SUBAPPLICATION Speed_Selection (* Waehlt aus den verfuegbaren Geschwindigkeitssignalen (VDS, WBSD, GBSD, MSS) das vom Bediener ausgewaehlte Signal aus und stellt Geschwindigkeit, Richtung und zurueckgelegte Distanz bereit; die Auswahl wird persistent im NVS gespeichert *)
  (* Standard: 61499-2 *)
  (* Version 1.0, 2025-04-01, Elias *)
  PACKAGE FBs::Baumsetzer::func::Automatik;
  IMPORT NVS_Keys::Key_GBSD_Store;
  IMPORT NVS_Keys::Key_MSS_Store;
  IMPORT NVS_Keys::Key_NMEA_Store;
  IMPORT NVS_Keys::Key_VDS_Store;
  IMPORT NVS_Keys::Key_WBSD_Store;
  IMPORT isobus::UT::Q::const::colours::COLOR_GREEN;
  IMPORT isobus::UT::Q::const::colours::COLOR_RED;
  IMPORT isobus::UT::io::Button::ButtonActivationCode::BT_RELEASED_UNLATCHED;
  IMPORT test::FBs::Baumsetzer::Constants::DefaultPool;
  IMPORT test::FBs::Baumsetzer::Constants::DefaultPool::Button_GBSD;
  IMPORT test::FBs::Baumsetzer::Constants::DefaultPool::Button_MSS;
  IMPORT test::FBs::Baumsetzer::Constants::DefaultPool::Button_NMEA;
  IMPORT test::FBs::Baumsetzer::Constants::DefaultPool::Button_VDS;
  IMPORT test::FBs::Baumsetzer::Constants::DefaultPool::Button_WBSD;
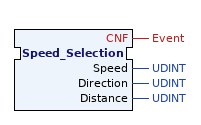
  EVENT_OUTPUT
    CNF; (* Execution Confirmation *)
  END_EVENT
  VAR_OUTPUT
    Speed : UDINT; (* Speed of selected Signal *)
    Direction : UDINT; (* Direction of selected Signal *)
    Distance : UDINT; (* Distance of selected Signal *)
  END_VAR
  FBS
    I_MSS : isobus::tecu::I_MSS(QI := FALSE);
    I_GBSD : isobus::tecu::I_GBSD(QI := FALSE);
    I_WBSD : isobus::tecu::I_WBSD(QI := FALSE);
    I_VDS : isobus::tecu::I_VDS(QI := FALSE);
    Button_VDS : isobus::UT::io::Button::Button_IE(QI := TRUE, u16ObjId := Button_VDS, InputEvent := BT_RELEASED_UNLATCHED);
    Button_WBSD : isobus::UT::io::Button::Button_IE(QI := TRUE, PARAMS := '', u16ObjId := Button_WBSD, InputEvent := BT_RELEASED_UNLATCHED);
    Button_GBSD : isobus::UT::io::Button::Button_IE(QI := TRUE, u16ObjId := Button_GBSD, InputEvent := BT_RELEASED_UNLATCHED);
    Button_MSS : isobus::UT::io::Button::Button_IE(QI := TRUE, u16ObjId := Button_MSS, InputEvent := BT_RELEASED_UNLATCHED);
    F_UINT_TO_REAL : iec61131::conversion::F_UINT_TO_REAL;
    CYCLE_TIME : logiBUS::utils::timing::CYCLE_TIME;
    INTEGRAL : logiBUS::utils::math::INTEGRAL;
    E_T_FF_SR : iec61499::events::E_T_FF_SR;
    E_T_FF_SR_1 : iec61499::events::E_T_FF_SR;
    E_T_FF_SR_2 : iec61499::events::E_T_FF_SR;
    E_T_FF_SR_3 : iec61499::events::E_T_FF_SR;
    F_SEL_E_Distance : eclipse4diac::utils::selection::F_SEL_E_4;
    F_SEL_E_Speed : eclipse4diac::utils::selection::F_SEL_E_4;
    F_SEL_E_Direction : eclipse4diac::utils::selection::F_SEL_E_4;
    COGSOGRapidUpdate : isobus::tecu::I_COGSOGRapidUpdate;
    E_T_FF_SR_4 : iec61499::events::E_T_FF_SR;
    Button_NMEA : isobus::UT::io::Button::Button_IE(QI := TRUE, u16ObjId := Button_NMEA, InputEvent := BT_RELEASED_UNLATCHED);
    INTEGRAL_1 : logiBUS::utils::math::INTEGRAL;
    CYCLE_TIME_1 : logiBUS::utils::timing::CYCLE_TIME;
    F_UINT_TO_REAL_1 : iec61131::conversion::F_UINT_TO_REAL;
    F_SEL_E_Distance_2 : eclipse4diac::utils::selection::F_SEL_E_2;
    F_SEL_E_Speed_2 : eclipse4diac::utils::selection::F_SEL_E_2;
    F_SEL_E_Direction_2 : eclipse4diac::utils::selection::F_SEL_E_2;
    UDINT2UDINT : iec61131::selection::F_MOVE; {SET_ATTRIBUTE(DataType, UDINT)}
    UDINT2UDINT_1 : iec61131::selection::F_MOVE; {SET_ATTRIBUTE(DataType, UDINT)}
    UDINT2UDINT_2 : iec61131::selection::F_MOVE; {SET_ATTRIBUTE(DataType, UDINT)}
    E_PERMIT : iec61499::events::E_PERMIT;
    E_PERMIT_1 : iec61499::events::E_PERMIT;
    E_PERMIT_2 : iec61499::events::E_PERMIT;
    E_PERMIT_4 : iec61499::events::E_PERMIT;
    F_SEL : iec61131::selection::F_SEL(IN0 := COLOR_RED, IN1 := COLOR_GREEN);
    Q_BackgroundColour : isobus::UT::Q::Q_BackgroundColour(u16ObjId := Button_VDS);
    Q_BackgroundColour_1 : isobus::UT::Q::Q_BackgroundColour(u16ObjId := Button_WBSD);
    F_SEL_1 : iec61131::selection::F_SEL(IN0 := COLOR_RED, IN1 := COLOR_GREEN);
    Q_BackgroundColour_2 : isobus::UT::Q::Q_BackgroundColour(u16ObjId := Button_GBSD);
    F_SEL_2 : iec61131::selection::F_SEL(IN0 := COLOR_RED, IN1 := COLOR_GREEN);
    Q_BackgroundColour_3 : isobus::UT::Q::Q_BackgroundColour(u16ObjId := Button_MSS);
    F_SEL_3 : iec61131::selection::F_SEL(IN0 := COLOR_RED, IN1 := COLOR_GREEN);
    Q_BackgroundColour_4 : isobus::UT::Q::Q_BackgroundColour(u16ObjId := Button_NMEA);
    F_SEL_4 : iec61131::selection::F_SEL(IN0 := COLOR_RED, IN1 := COLOR_GREEN);
    Geschwindigkeit : isobus::UT::Q::Q_NumericValue(u16ObjId := DefaultPool::OutputNumber_12000);
    Geschwindigkeit_1 : isobus::UT::Q::Q_NumericValue(u16ObjId := DefaultPool::OutputNumber_12004);
    Geschwindigkeit_2 : isobus::UT::Q::Q_NumericValue(u16ObjId := DefaultPool::OutputNumber_12005);
    Geschwindigkeit_3 : isobus::UT::Q::Q_NumericValue(u16ObjId := DefaultPool::OutputNumber_12006);
    Geschwindigkeit_4 : isobus::UT::Q::Q_NumericValue(u16ObjId := DefaultPool::OutputNumber_12007);
    F_MUL : iec61131::arithmetic::F_MUL(IN2 := uint#10);
    CYCLE_TIME_2 : logiBUS::utils::timing::CYCLE_TIME;
    E_PERMIT_5 : iec61499::events::E_PERMIT;
    INTEGRAL_2 : logiBUS::utils::math::INTEGRAL;
    F_UINT_TO_REAL_2 : iec61131::conversion::F_UINT_TO_REAL;
    F_REAL_TO_UDINT : iec61131::conversion::F_REAL_TO_UDINT;
    F_REAL_TO_UDINT_1 : iec61131::conversion::F_REAL_TO_UDINT;
    F_REAL_TO_UDINT_2 : iec61131::conversion::F_REAL_TO_UDINT;
    UDINT2UDINT_Distance : iec61131::selection::F_MOVE; {SET_ATTRIBUTE(DataType, UDINT)}
    UDINT2UDINT_Speed : iec61131::selection::F_MOVE; {SET_ATTRIBUTE(DataType, UDINT)}
    UDINT2UDINT_Direction : iec61131::selection::F_MOVE; {SET_ATTRIBUTE(DataType, UDINT)}
    VDS_Selected : logiBUS::storage::esp32_nvs::NVS(QI := TRUE, KEY := Key_VDS_Store, DEFAULT_VALUE := bool#FALSE);
    WBSD_Selected : logiBUS::storage::esp32_nvs::NVS(QI := TRUE, KEY := Key_WBSD_Store, DEFAULT_VALUE := bool#TRUE);
    GBSD_Selected : logiBUS::storage::esp32_nvs::NVS(QI := TRUE, KEY := Key_GBSD_Store, DEFAULT_VALUE := bool#FALSE);
    F_MOVE_2 : iec61131::selection::F_MOVE; {SET_ATTRIBUTE(DataType, BOOL)}
    MSS_Selected : logiBUS::storage::esp32_nvs::NVS(QI := TRUE, KEY := Key_MSS_Store, DEFAULT_VALUE := bool#FALSE);
    F_MOVE_3 : iec61131::selection::F_MOVE; {SET_ATTRIBUTE(DataType, BOOL)}
    NMEA_Selected : logiBUS::storage::esp32_nvs::NVS(QI := TRUE, KEY := Key_NMEA_Store, DEFAULT_VALUE := bool#FALSE);
    F_MOVE_4 : iec61131::selection::F_MOVE; {SET_ATTRIBUTE(DataType, BOOL)}
    F_MOVE : iec61131::selection::F_MOVE; {SET_ATTRIBUTE(DataType, BOOL)}
    F_MOVE_1 : iec61131::selection::F_MOVE; {SET_ATTRIBUTE(DataType, BOOL)}
    F_MOVE_5 : iec61131::selection::F_MOVE; {SET_ATTRIBUTE(DataType, UINT)}
  END_FBS
  EVENT_CONNECTIONS
    I_VDS.IND TO F_UINT_TO_REAL.REQ;
    I_VDS.IND TO CYCLE_TIME.REQ;
    F_UINT_TO_REAL.CNF TO INTEGRAL.REQ;
    Button_VDS.IND TO E_T_FF_SR.S;
    Button_WBSD.IND TO E_T_FF_SR.R;
    Button_GBSD.IND TO E_T_FF_SR.R;
    Button_MSS.IND TO E_T_FF_SR.R;
    Button_WBSD.IND TO E_T_FF_SR_1.S;
    Button_VDS.IND TO E_T_FF_SR_1.R;
    Button_GBSD.IND TO E_T_FF_SR_1.R;
    Button_MSS.IND TO E_T_FF_SR_1.R;
    Button_GBSD.IND TO E_T_FF_SR_2.S;
    Button_MSS.IND TO E_T_FF_SR_2.R;
    Button_WBSD.IND TO E_T_FF_SR_2.R;
    Button_VDS.IND TO E_T_FF_SR_2.R;
    Button_MSS.IND TO E_T_FF_SR_3.S;
    Button_GBSD.IND TO E_T_FF_SR_3.R;
    Button_WBSD.IND TO E_T_FF_SR_3.R;
    Button_VDS.IND TO E_T_FF_SR_3.R;
    Button_WBSD.IND TO E_T_FF_SR_4.R;
    Button_VDS.IND TO E_T_FF_SR_4.R;
    Button_GBSD.IND TO E_T_FF_SR_4.R;
    Button_MSS.IND TO E_T_FF_SR_4.R;
    Button_NMEA.IND TO E_T_FF_SR_1.R;
    Button_NMEA.IND TO E_T_FF_SR_4.S;
    Button_NMEA.IND TO E_T_FF_SR_2.R;
    Button_NMEA.IND TO E_T_FF_SR.R;
    Button_NMEA.IND TO E_T_FF_SR_3.R;
    F_UINT_TO_REAL_1.CNF TO INTEGRAL_1.REQ;
    F_SEL_E_Distance.CNF TO UDINT2UDINT.REQ;
    UDINT2UDINT.CNF TO F_SEL_E_Distance_2.REQ1;
    F_SEL_E_Speed.CNF TO UDINT2UDINT_1.REQ;
    UDINT2UDINT_1.CNF TO F_SEL_E_Speed_2.REQ1;
    F_SEL_E_Direction.CNF TO UDINT2UDINT_2.REQ;
    UDINT2UDINT_2.CNF TO F_SEL_E_Direction_2.REQ1;
    F_MOVE_2.CNF TO I_GBSD.INIT;
    F_MOVE_3.CNF TO I_MSS.INIT;
    F_MOVE_4.CNF TO COGSOGRapidUpdate.INIT;
    E_PERMIT.EO TO F_SEL_E_Distance.REQ1;
    INTEGRAL.CNF TO E_PERMIT.EI;
    E_PERMIT.EO TO F_SEL_E_Speed.REQ1;
    E_PERMIT.EO TO F_SEL_E_Direction.REQ1;
    I_WBSD.IND TO E_PERMIT_1.EI;
    E_PERMIT_1.EO TO F_SEL_E_Distance.REQ2;
    E_PERMIT_1.EO TO F_SEL_E_Direction.REQ2;
    E_PERMIT_1.EO TO F_SEL_E_Speed.REQ2;
    I_GBSD.IND TO E_PERMIT_2.EI;
    E_PERMIT_2.EO TO F_SEL_E_Distance.REQ3;
    E_PERMIT_2.EO TO F_SEL_E_Speed.REQ3;
    E_PERMIT_2.EO TO F_SEL_E_Direction.REQ3;
    INTEGRAL_1.CNF TO E_PERMIT_4.EI;
    E_PERMIT_4.EO TO F_SEL_E_Direction_2.REQ2;
    E_PERMIT_4.EO TO F_SEL_E_Distance_2.REQ2;
    E_PERMIT_4.EO TO F_SEL_E_Speed_2.REQ2;
    F_SEL.CNF TO Q_BackgroundColour.REQ;
    F_SEL_1.CNF TO Q_BackgroundColour_1.REQ;
    F_SEL_2.CNF TO Q_BackgroundColour_2.REQ;
    F_SEL_3.CNF TO Q_BackgroundColour_3.REQ;
    F_SEL_4.CNF TO Q_BackgroundColour_4.REQ;
    F_MOVE_2.CNF TO F_SEL_2.REQ;
    F_MOVE_3.CNF TO F_SEL_3.REQ;
    F_MOVE_4.CNF TO F_SEL_4.REQ;
    I_WBSD.IND TO Geschwindigkeit.REQ;
    I_VDS.IND TO Geschwindigkeit_1.REQ;
    I_GBSD.IND TO Geschwindigkeit_2.REQ;
    I_MSS.IND TO Geschwindigkeit_3.REQ;
    COGSOGRapidUpdate.IND TO F_MUL.REQ;
    F_MOVE_5.CNF TO CYCLE_TIME_1.REQ;
    F_MOVE_5.CNF TO F_UINT_TO_REAL_1.REQ;
    F_MOVE_5.CNF TO Geschwindigkeit_4.REQ;
    F_UINT_TO_REAL_2.CNF TO INTEGRAL_2.REQ;
    INTEGRAL_2.CNF TO E_PERMIT_5.EI;
    I_MSS.IND TO F_UINT_TO_REAL_2.REQ;
    I_MSS.IND TO CYCLE_TIME_2.REQ;
    E_PERMIT_5.EO TO F_SEL_E_Direction.REQ4;
    E_PERMIT_5.EO TO F_SEL_E_Speed.REQ4;
    E_PERMIT_5.EO TO F_SEL_E_Distance.REQ4;
    E_PERMIT.EO TO F_REAL_TO_UDINT.REQ;
    E_PERMIT_5.EO TO F_REAL_TO_UDINT_1.REQ;
    E_PERMIT_4.EO TO F_REAL_TO_UDINT_2.REQ;
    F_SEL_E_Distance_2.CNF TO UDINT2UDINT_Distance.REQ;
    UDINT2UDINT_Speed.CNF TO CNF;
    F_SEL_E_Speed_2.CNF TO UDINT2UDINT_Speed.REQ;
    F_SEL_E_Direction_2.CNF TO UDINT2UDINT_Direction.REQ;
    E_T_FF_SR.EO TO VDS_Selected.SET;
    E_T_FF_SR_1.EO TO WBSD_Selected.SET;
    E_T_FF_SR_2.EO TO GBSD_Selected.SET;
    GBSD_Selected.SETO TO F_MOVE_2.REQ;
    GBSD_Selected.GETO TO F_MOVE_2.REQ;
    MSS_Selected.SETO TO F_MOVE_3.REQ;
    MSS_Selected.GETO TO F_MOVE_3.REQ;
    E_T_FF_SR_3.EO TO MSS_Selected.SET;
    E_T_FF_SR_4.EO TO NMEA_Selected.SET;
    NMEA_Selected.GETO TO F_MOVE_4.REQ;
    NMEA_Selected.SETO TO F_MOVE_4.REQ;
    VDS_Selected.SETO TO F_MOVE.REQ;
    VDS_Selected.GETO TO F_MOVE.REQ;
    F_MOVE.CNF TO I_VDS.INIT;
    F_MOVE.CNF TO F_SEL.REQ;
    WBSD_Selected.SETO TO F_MOVE_1.REQ;
    WBSD_Selected.GETO TO F_MOVE_1.REQ;
    F_MOVE_1.CNF TO I_WBSD.INIT;
    F_MOVE_1.CNF TO F_SEL_1.REQ;
    F_MUL.CNF TO F_MOVE_5.REQ;
  END_CONNECTIONS
  DATA_CONNECTIONS
    I_VDS.NavigationBasedVehicleSpeed TO F_UINT_TO_REAL.IN;
    I_VDS.timestamp_data TO CYCLE_TIME.TM;
    F_UINT_TO_REAL.OUT TO INTEGRAL.IN;
    CYCLE_TIME.CYCLE TO INTEGRAL.TM;
    F_MOVE_3.OUT TO I_MSS.QI;
    F_MOVE_2.OUT TO I_GBSD.QI;
    I_WBSD.WHEELBASEDMACHINEDISTANCE TO F_SEL_E_Distance.IN2;
    I_GBSD.GROUNDBASEDMACHINEDISTANCE TO F_SEL_E_Distance.IN3;
    I_VDS.NavigationBasedVehicleSpeed TO F_SEL_E_Speed.IN1;
    I_WBSD.WHEELBASEDMACHINESPEED TO F_SEL_E_Speed.IN2;
    I_GBSD.GROUNDBASEDMACHINESPEED TO F_SEL_E_Speed.IN3;
    I_MSS.SELECTEDMACHINESPEED TO F_SEL_E_Speed.IN4;
    I_MSS.SELECTEDMACHINEDIRECTION TO F_SEL_E_Direction.IN4;
    I_GBSD.GROUNDBASEDMACHINEDIRECTION TO F_SEL_E_Direction.IN3;
    I_WBSD.WHEELBASEDMACHINEDIRECTION TO F_SEL_E_Direction.IN2;
    F_MOVE_4.OUT TO COGSOGRapidUpdate.QI;
    CYCLE_TIME_1.CYCLE TO INTEGRAL_1.TM;
    F_UINT_TO_REAL_1.OUT TO INTEGRAL_1.IN;
    COGSOGRapidUpdate.timestamp_data TO CYCLE_TIME_1.TM;
    F_SEL_E_Distance.OUT TO UDINT2UDINT.IN;
    F_SEL_E_Speed.OUT TO UDINT2UDINT_1.IN;
    UDINT2UDINT_1.OUT TO F_SEL_E_Speed_2.IN1;
    COGSOGRapidUpdate.SpeedOverGround TO F_SEL_E_Speed_2.IN2;
    F_SEL_E_Direction.OUT TO UDINT2UDINT_2.IN;
    UDINT2UDINT_2.OUT TO F_SEL_E_Direction_2.IN1;
    I_WBSD.WHEELBASEDMACHINEDIRECTION TO F_SEL_E_Direction.IN1;
    I_WBSD.WHEELBASEDMACHINEDIRECTION TO F_SEL_E_Direction_2.IN2;
    F_MOVE_2.OUT TO E_PERMIT_2.PERMIT;
    F_MOVE_4.OUT TO E_PERMIT_4.PERMIT;
    F_SEL.OUT TO Q_BackgroundColour.u8Colour;
    F_SEL_1.OUT TO Q_BackgroundColour_1.u8Colour;
    F_MOVE_2.OUT TO F_SEL_2.G;
    F_SEL_2.OUT TO Q_BackgroundColour_2.u8Colour;
    F_SEL_3.OUT TO Q_BackgroundColour_3.u8Colour;
    F_MOVE_3.OUT TO F_SEL_3.G;
    F_SEL_4.OUT TO Q_BackgroundColour_4.u8Colour;
    F_MOVE_4.OUT TO F_SEL_4.G;
    I_WBSD.WHEELBASEDMACHINESPEED TO Geschwindigkeit.u32NewValue;
    I_VDS.NavigationBasedVehicleSpeed TO Geschwindigkeit_1.u32NewValue;
    I_GBSD.GROUNDBASEDMACHINESPEED TO Geschwindigkeit_2.u32NewValue;
    I_MSS.SELECTEDMACHINESPEED TO Geschwindigkeit_3.u32NewValue;
    COGSOGRapidUpdate.SpeedOverGround TO F_MUL.IN1;
    F_MOVE_5.OUT TO F_UINT_TO_REAL_1.IN;
    F_MOVE_5.OUT TO Geschwindigkeit_4.u32NewValue;
    CYCLE_TIME_2.CYCLE TO INTEGRAL_2.TM;
    F_UINT_TO_REAL_2.OUT TO INTEGRAL_2.IN;
    I_MSS.timestamp_data TO CYCLE_TIME_2.TM;
    I_MSS.SELECTEDMACHINESPEED TO F_UINT_TO_REAL_2.IN;
    F_MOVE_3.OUT TO E_PERMIT_5.PERMIT;
    INTEGRAL.OUT TO F_REAL_TO_UDINT.IN;
    INTEGRAL_2.OUT TO F_REAL_TO_UDINT_1.IN;
    F_REAL_TO_UDINT_1.OUT TO F_SEL_E_Distance.IN4;
    INTEGRAL_1.OUT TO F_REAL_TO_UDINT_2.IN;
    F_REAL_TO_UDINT_2.OUT TO F_SEL_E_Distance_2.IN2;
    F_SEL_E_Distance_2.OUT TO UDINT2UDINT_Distance.IN;
    UDINT2UDINT_Speed.OUT TO Speed;
    UDINT2UDINT_Direction.OUT TO Direction;
    UDINT2UDINT_Distance.OUT TO Distance;
    F_SEL_E_Speed_2.OUT TO UDINT2UDINT_Speed.IN;
    F_SEL_E_Direction_2.OUT TO UDINT2UDINT_Direction.IN;
    E_T_FF_SR.Q TO VDS_Selected.VALUE;
    E_T_FF_SR_1.Q TO WBSD_Selected.VALUE;
    E_T_FF_SR_2.Q TO GBSD_Selected.VALUE;
    GBSD_Selected.VALUEO TO F_MOVE_2.IN;
    MSS_Selected.VALUEO TO F_MOVE_3.IN;
    E_T_FF_SR_3.Q TO MSS_Selected.VALUE;
    E_T_FF_SR_4.Q TO NMEA_Selected.VALUE;
    NMEA_Selected.VALUEO TO F_MOVE_4.IN;
    F_REAL_TO_UDINT.OUT TO F_SEL_E_Distance.IN1;
    UDINT2UDINT.OUT TO F_SEL_E_Distance_2.IN1;
    VDS_Selected.VALUEO TO F_MOVE.IN;
    F_MOVE.OUT TO E_PERMIT.PERMIT;
    F_MOVE.OUT TO F_SEL.G;
    WBSD_Selected.VALUEO TO F_MOVE_1.IN;
    F_MOVE_1.OUT TO I_WBSD.QI;
    F_MOVE.OUT TO I_VDS.QI;
    F_MOVE_1.OUT TO E_PERMIT_1.PERMIT;
    F_MOVE_1.OUT TO F_SEL_1.G;
    F_MUL.OUT TO F_MOVE_5.IN;
  END_CONNECTIONS
END_SUBAPPLICATION
